FUNCTION_BLOCK PID_CALC
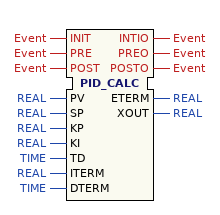
  EVENT_INPUT
    INIT;
    PRE;
    POST;
  END_EVENT
  EVENT_OUTPUT
    INTIO;
    PREO;
    POSTO;
  END_EVENT
  VAR_INPUT
    PV : REAL;
    SP : REAL;
    KP : REAL;
    KI : REAL;
    TD : TIME;
    ITERM : REAL;
    DTERM : TIME;
  END_VAR
  VAR_OUTPUT
    ETERM : REAL;
    XOUT : REAL;
  END_VAR
  EC_STATES
    START;
  END_STATES
END_FUNCTION_BLOCK
